Staubli VAL3: getSize.pgx

public program getSize(num& x_nSize[])
begin
  //
  // get the size of the list
  //
end
